
// ===== library: MasterCopy "Kopie von Programmbausteine in GW_Materialparameter" =====

// folder: GW_Materialparameter

DATA_BLOCK "DB_GW_Materialparameter"   // DB241
{ S7_Optimized_Access := 'TRUE' }
VERSION : 0.1
   VAR
      Gewerk_1 : "UDT_GW_Gewerk_1";
      Gewerk_2 : "UDT_GW_Gewerk_2";
      Gesamt_gueltig : Bool;   // Gesamt gültig
      Gesamt_differenz : Bool;   // Gesamt differenz
      Gesamt_uebernehmen : Bool;   // Gesamt übernehmen
      Gesamt_verwerfen : Bool;   // Gesamt verwerfen
   END_VAR
BEGIN
END_DATA_BLOCK

FUNCTION "FC_GW_Materialparameter" : Void   // FC37, FBD
{ S7_Optimized_Access := 'TRUE' }
VERSION : 0.1
   VAR_IN_OUT
      Gewerk_1 : "UDT_GW_Gewerk_1";
      Gewerk_2 : "UDT_GW_Gewerk_2";
   END_VAR
BEGIN

REGION Network 1: Sollwerte Grenzen prüfen
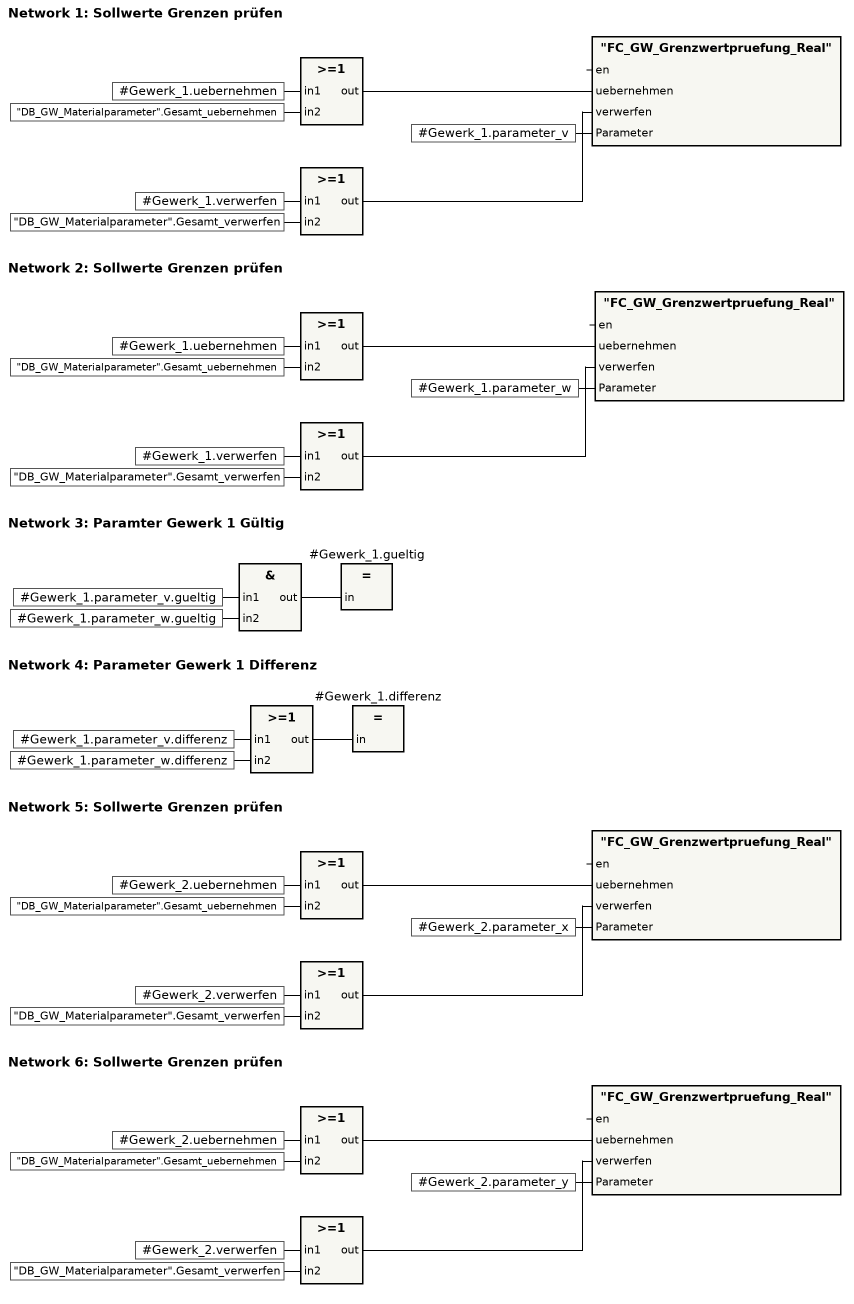
   "FC_GW_Grenzwertpruefung_Real"(uebernehmen := #Gewerk_1.uebernehmen OR "DB_GW_Materialparameter".Gesamt_uebernehmen,
                           verwerfen := #Gewerk_1.verwerfen OR "DB_GW_Materialparameter".Gesamt_verwerfen,
                           Parameter := #Gewerk_1.parameter_v);
END_REGION

REGION Network 2: Sollwerte Grenzen prüfen
   "FC_GW_Grenzwertpruefung_Real"(uebernehmen := #Gewerk_1.uebernehmen OR "DB_GW_Materialparameter".Gesamt_uebernehmen,
                           verwerfen := #Gewerk_1.verwerfen OR "DB_GW_Materialparameter".Gesamt_verwerfen,
                           Parameter := #Gewerk_1.parameter_w);
END_REGION

REGION Network 3: Paramter Gewerk 1 Gültig
   #Gewerk_1.gueltig := #Gewerk_1.parameter_v.gueltig AND #Gewerk_1.parameter_w.gueltig;
END_REGION

REGION Network 4: Parameter Gewerk 1 Differenz
   #Gewerk_1.differenz := #Gewerk_1.parameter_v.differenz OR #Gewerk_1.parameter_w.differenz;
END_REGION

REGION Network 5: Sollwerte Grenzen prüfen
   "FC_GW_Grenzwertpruefung_Real"(uebernehmen := #Gewerk_2.uebernehmen OR "DB_GW_Materialparameter".Gesamt_uebernehmen,
                           verwerfen := #Gewerk_2.verwerfen OR "DB_GW_Materialparameter".Gesamt_verwerfen,
                           Parameter := #Gewerk_2.parameter_x);
END_REGION

REGION Network 6: Sollwerte Grenzen prüfen
   "FC_GW_Grenzwertpruefung_Real"(uebernehmen := #Gewerk_2.uebernehmen OR "DB_GW_Materialparameter".Gesamt_uebernehmen,
                           verwerfen := #Gewerk_2.verwerfen OR "DB_GW_Materialparameter".Gesamt_verwerfen,
                           Parameter := #Gewerk_2.parameter_y);
END_REGION

REGION Network 7: Sollwerte Grenzen prüfen
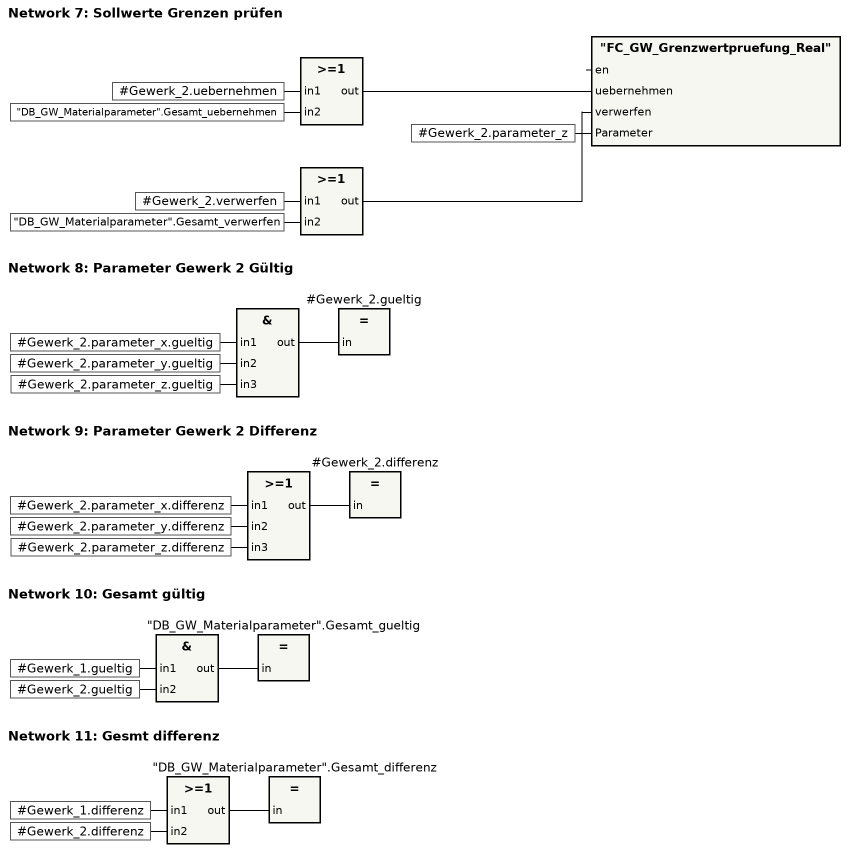
   "FC_GW_Grenzwertpruefung_Real"(uebernehmen := #Gewerk_2.uebernehmen OR "DB_GW_Materialparameter".Gesamt_uebernehmen,
                           verwerfen := #Gewerk_2.verwerfen OR "DB_GW_Materialparameter".Gesamt_verwerfen,
                           Parameter := #Gewerk_2.parameter_z);
END_REGION

REGION Network 8: Parameter Gewerk 2 Gültig
   #Gewerk_2.gueltig := #Gewerk_2.parameter_x.gueltig AND #Gewerk_2.parameter_y.gueltig AND #Gewerk_2.parameter_z.gueltig;
END_REGION

REGION Network 9: Parameter Gewerk 2 Differenz
   #Gewerk_2.differenz := #Gewerk_2.parameter_x.differenz OR #Gewerk_2.parameter_y.differenz OR #Gewerk_2.parameter_z.differenz;
END_REGION

REGION Network 10: Gesamt gültig
   "DB_GW_Materialparameter".Gesamt_gueltig := #Gewerk_1.gueltig AND #Gewerk_2.gueltig;
END_REGION

REGION Network 11: Gesmt differenz
   "DB_GW_Materialparameter".Gesamt_differenz := #Gewerk_1.differenz OR #Gewerk_2.differenz;
END_REGION

REGION Network 12 (SCL): Übernehmen und Verwerfen rücksetzen
   #Gewerk_1.uebernehmen:= FALSE;
   #Gewerk_1.verwerfen:= FALSE;
   #Gewerk_2.uebernehmen:= FALSE;
   #Gewerk_2.verwerfen:= FALSE;
   "DB_GW_Materialparameter".Gesamt_uebernehmen:= FALSE;
   "DB_GW_Materialparameter".Gesamt_verwerfen:= FALSE;
END_REGION
END_FUNCTION

FUNCTION "FC_GW_Grenzwertpruefung_Real" : Void   // FC38, FBD
{ S7_Optimized_Access := 'TRUE' }
VERSION : 0.1
   VAR_INPUT
      uebernehmen : Bool;
      verwerfen : Bool;
   END_VAR
   VAR_IN_OUT
      Parameter : "UDT_GW_Parameter";
   END_VAR
BEGIN

REGION Network 1 (SCL): Gueltig
   IF #Parameter.wert > #Parameter.max OR
       #Parameter.wert < #Parameter.min THEN
       #Parameter.gueltig:= FALSE;
   ELSE
       #Parameter.gueltig:= TRUE;
   END_IF;
END_REGION

REGION Network 2 (SCL): Differenz zwischen Aktiv
   IF #Parameter.wert <> #Parameter.wert_aktiv THEN
       #Parameter.differenz:= TRUE;
   ELSE
       #Parameter.differenz:= FALSE;
   END_IF;
END_REGION

REGION Network 3 (SCL): Übernehmen Verwerfen
   IF #Parameter.gueltig AND #uebernehmen THEN
       #Parameter.wert_aktiv:= #Parameter.wert;
   END_IF;

   IF #verwerfen THEN
       #Parameter.wert:= #Parameter.wert_aktiv;
   END_IF;
END_REGION
END_FUNCTION

// ===== library: MasterCopy "UDT_GW_Gewerk_1" =====

TYPE "UDT_GW_Gewerk_1"
   STRUCT
      parameter_v : "UDT_GW_Parameter";
      parameter_w : "UDT_GW_Parameter";
      gueltig : Bool;   // Gewerk gültig
      differenz : Bool;   // Gewerk differenz zu Aktiv
      uebernehmen : Bool;   // Gewerk übernehmen
      verwerfen : Bool;   // Gewerk verwerfen
   END_STRUCT;
END_TYPE

// ===== library: MasterCopy "UDT_GW_Gewerk_2" =====

TYPE "UDT_GW_Gewerk_2"
   STRUCT
      parameter_x : "UDT_GW_Parameter";
      parameter_y : "UDT_GW_Parameter";
      parameter_z : "UDT_GW_Parameter";
      gueltig : Bool;   // Gewerk gültig
      differenz : Bool;   // Gewerk differenz zu Aktiv
      uebernehmen : Bool;   // Gewerk übernehmen
      verwerfen : Bool;   // Gewerk verwerfen
   END_STRUCT;
END_TYPE

// ===== library: MasterCopy "UDT_GW_Parameter" =====

TYPE "UDT_GW_Parameter"
   STRUCT
      wert : Real;   // Parameterwert der auf der Visu eingegeben wird
      wert_aktiv : Real;   // Parameterwert mit dem die Anlage arbeitet
      min : Real;   // Min Begrenzung
      max : Real;   // Max Begrenzung
      gueltig : Bool;   // Eingabewert Befindet sich innerhalb der Grenzwerte Min Max
      differenz : Bool;   // Differenz zu aktiv
   END_STRUCT;
END_TYPE